{attribute 'linkalways'} 
{attribute 'no_explicit_call' := 'This FB is a CLASS and must be accessed using methods or properties'}
{attribute 'enable_dynamic_creation'}
FUNCTION_BLOCK Node_F_VN_ImageCenterOfMass EXTENDS VisionNode
VAR
    ipSrcImage : _ITcVnImage;
    aCenterOfMass : _TcVnPoint2_LREAL;
    hrPrev : _HRESULT(S_OK);
	hresult : _HRESULT(S_OK);
END_VAR

METHOD PUBLIC  Clone : I_Node
VAR
	pNode : POINTER TO Node_F_VN_ImageCenterOfMass;
END_VAR
pNode := __NEW(Node_F_VN_ImageCenterOfMass);
Clone := pNode^;
END_METHOD

METHOD FB_init : BOOL
VAR_INPUT
	bInitRetains : BOOL; // if TRUE, the retain variables are initialized (warm start / cold start)
	bInCopyCode : BOOL;  // if TRUE, the instance afterwards gets moved into the copy code (online change)
END_VAR
AddInput('ipSrcImage', ipSrcImage);
AddInput('hrPrev', hrPrev);
AddOutput('aCenterOfMass', aCenterOfMass);
AddOutput('hresult', hresult);
END_METHOD

METHOD PROTECTED OnExecute
hresult.Value := F_VN_ImageCenterOfMass(
	ipSrcImage := ipSrcImage.Value,
    aCenterOfMass := aCenterOfMass.Value,
	hrPrev:= hrPrev.Value);
END_METHOD

METHOD PUBLIC PreExecutionCheck
VAR_INPUT
	Check : I_PreExecutionChecks;
END_VAR
Check.IsTrue(ipSrcImage.IsValid, 'ipSrcImage must contain an image');
Check.IsTrue(ipSrcImage.HasChannelCount(1), 'ipSrcImage must contain 1 channel');
END_METHOD

END_FUNCTION_BLOCK

(* stored: Version 1.1.0.1, ProductVersion 3.1.4024.13
   POU Node_F_VN_ImageCenterOfMass: Id {3ca14467-fa76-03e1-0f0d-651ef8f84649}, SpecialFunc None
   Folder Constructor: Id {792022da-eaf2-0c3c-34ce-fa4553f88c89}
   Method Clone: Id {44cd8c4c-1196-0c0a-1044-638dce24fad6}
   Method FB_init: Id {657b60df-cd7b-009d-0203-8dbceb8fdfa3}
   Method OnExecute: Id {9cf882df-b695-0e4d-19cb-8fe58c07f057}
   Method PreExecutionCheck: Id {d45c37b0-d9f3-023d-27a6-93cae9f81338} *)
